MOVL C09996 V=800.0 PL=0
CALL JOB:A_ROOF_SIDE_0617_2_PAINT_5
END
